// TwinCAT 3 PLC project PLC1
// ProgramVersion: 3.1.4023.0
// libraries:
//   Tc2_Standard, * (Beckhoff Automation GmbH)
//   Tc2_System, * (Beckhoff Automation GmbH)
//   Tc2_Utilities, * (Beckhoff Automation GmbH)
//   Tc3_IotBase, * (Beckhoff Automation GmbH)
//   Tc3_JsonXml, * (Beckhoff Automation GmbH)
//   Tc3_Module, * (Beckhoff Automation GmbH)
// project tree:
//   DUTs/ ST_INSUMOS.TcDUT (not stored)
//   / PlcTask.TcTTO (not stored)
//   POUs/ CheckBounds.TcPOU, CheckDivDInt.TcPOU (not stored), CheckDivLInt.TcPOU (not stored), CheckDivLReal.TcPOU, CheckDivReal.TcPOU (not stored), CheckLRangeSigned.TcPOU, CheckLRangeUnsigned.TcPOU, CheckPointer.TcPOU, CheckRangeSigned.TcPOU (not stored), CheckRangeUnsigned.TcPOU (not stored), MAIN.TcPOU
//   POUs/HTTP/ FB_ParseString.TcPOU (not stored), FB_TestHTTP_Get.TcPOU, FB_TestHTTP_HeaderAuth.TcPOU (not stored), FB_TestHTTP_Post.TcPOU (not stored), FB_TestHTTP_Put.TcPOU (not stored)

// ---- POUs/CheckBounds.TcPOU
// Implicitly generated code : DO NOT EDIT
FUNCTION CheckBounds : DINT
VAR_INPUT
	index, lower, upper: DINT;
END_VAR

// Implicitly generated code : Only an Implementation suggestion
{noflow}
IF  index < lower THEN
	CheckBounds := lower;
ELSIF  index > upper THEN
	CheckBounds := upper;
ELSE  
	CheckBounds := index;
END_IF
{flow}

END_FUNCTION

// ---- POUs/CheckDivLReal.TcPOU
// Implicitly generated code : DO NOT EDIT
FUNCTION CheckDivLReal : LREAL
VAR_INPUT
	divisor:LREAL;
END_VAR

// Implicitly generated code : Only an Implementation suggestion
{noflow}
IF divisor = 0 THEN
	CheckDivLReal:=1;
ELSE
	CheckDivLReal:=divisor;
END_IF;
{flow}

END_FUNCTION

// ---- POUs/CheckLRangeSigned.TcPOU
// Implicitly generated code : DO NOT EDIT
FUNCTION CheckLRangeSigned : LINT
VAR_INPUT
	value, lower, upper: LINT;
END_VAR

// Implicitly generated code : Only an Implementation suggestion
{noflow}
IF (value < lower) THEN
	CheckLRangeSigned := lower;
ELSIF(value > upper) THEN
	CheckLRangeSigned := upper;
ELSE
	CheckLRangeSigned := value;
END_IF

{flow}

END_FUNCTION

// ---- POUs/CheckLRangeUnsigned.TcPOU
// Implicitly generated code : DO NOT EDIT
FUNCTION CheckLRangeUnsigned : ULINT
VAR_INPUT
	value, lower, upper: ULINT;
END_VAR

// Implicitly generated code : Only an Implementation suggestion
{noflow}
IF (value < lower) THEN
	CheckLRangeUnsigned := lower;
ELSIF(value > upper) THEN
	CheckLRangeUnsigned := upper;
ELSE
	CheckLRangeUnsigned := value;
END_IF
{flow}

END_FUNCTION

// ---- POUs/CheckPointer.TcPOU
// Implicitly generated code : DO NOT EDIT
FUNCTION CheckPointer : POINTER TO BYTE
VAR_INPUT 
	ptToTest : POINTER TO BYTE; // Destination address of the pointer
	iSize : DINT;		        // Size of the type the pointer points to. (e.g: 20 for POINTER TO ARRAY [0..9] OF INT) 
	iGran : DINT;		        // Granularity of the pointer access. This is the size of the biggest non-structured data type in the type the pointer points to. (e.g: 2 for POINTER TO ARRAY [0..9] OF INT)
	bWrite: BOOL;		        // Indicates read or write Access. TRUE = write access.
END_VAR

// Implicitly generated code : Only an Implementation suggestion
{noflow}
IF ptToTest=0 THEN
    ADSLOGSTR(ADSLOG_MSGTYPE_ERROR OR ADSLOG_MSGTYPE_STRING,'CheckPointer failed due to invalid address.','');
ELSIF iSize<=0 THEN
    ADSLOGSTR(ADSLOG_MSGTYPE_ERROR OR ADSLOG_MSGTYPE_STRING,'CheckPointer failed due to invalid size.','');
ELSIF iGran<=0 THEN
    ADSLOGSTR(ADSLOG_MSGTYPE_ERROR OR ADSLOG_MSGTYPE_STRING,'CheckPointer failed due to invalid granularity.','');
// -> Please note that the following memory area check is time consuming:
//ELSIF F_CheckMemoryArea(pData:=ptToTest,nSize:=DINT_TO_UDINT(iSize)) = E_TcMemoryArea.Unknown THEN
//    ADSLOGSTR(ADSLOG_MSGTYPE_ERROR OR ADSLOG_MSGTYPE_STRING,'CheckPointer failed due to unknown memory area.','');
END_IF
CheckPointer := ptToTest;
{flow}

END_FUNCTION

// ---- POUs/MAIN.TcPOU
PROGRAM MAIN
VAR
	fbHttpClientPostman			: FB_IotHttpClient := (sHostName := '10.1.1.220',bKeepAlive:=TRUE);	
	fbHttpHeaderAuth			: FB_TestHTTP_HeaderAuth;
	
	bHeaderAuth 				: BOOL;
	bConvertBack				: BOOL;
	fbJsonDataType				: FB_JsonReadWriteDatatype;
	
	fbJson     : FB_JsonDomParser;
  		jsonProp   : SJsonValue;
  		jsonValue  : SJsonValue;
		
	bHasMember				: BOOL;
	operadorEncerrouLote	: DINT;
	data					: STRING(5000);
	insumos					: STRING(5000);
	arraySize				: UDINT;
	jsonIterator			: SJsonValue;
	jsonIteratorEnd			: SJsonValue;
	jsonIterator2			: SJsonValue;
	jsonIteratorEnd2		: SJsonValue;
	jsonIterator3			: SJsonValue;
	jsonIteratorEnd3		: SJsonValue;
	sName					: SJsonValue;
	jsonRoot				: SJsonValue;
	jsonRootInsumos			: SJsonValue;
	jsonRootInsumosDados	: SJsonValue;
	
	sTest:STRING(5000)		:= '{"continuationToken":"","data":[{"Insumos":[{"continuationToken":"","dados":[{"bloqueiaTerc":null,"centroCusto":"1011201002","classificacao":"1","classificacaoOrigem":"2","engenharia":"0201010080-0","insumo":"202010158","kanban":false,"natureza":"3","possuiAlternativos":false,"quantidadeTotal":"20000000","seqConsumo":4,"seqOperacao":1,"tipoInsumo":"1","transacaoBaixaEstoque":31},{"bloqueiaTerc":null,"centroCusto":"1011201002","classificacao":"1","classificacaoOrigem":"2","engenharia":"0201010080-0","insumo":"204010081","kanban":false,"natureza":"3","possuiAlternativos":false,"quantidadeTotal":"20000000","seqConsumo":2,"seqOperacao":1,"tipoInsumo":"1","transacaoBaixaEstoque":31},{"bloqueiaTerc":null,"centroCusto":"1011201002","classificacao":"1","classificacaoOrigem":"2","engenharia":"0201010080-0","insumo":"205050005","kanban":false,"natureza":"3","possuiAlternativos":false,"quantidadeTotal":"20000000","seqConsumo":3,"seqOperacao":1,"tipoInsumo":"1","transacaoBaixaEstoque":31}]}],"Lotes":[{"OperadorEncerrouLote":"163","codLote":"1-1","codOF":71605,"dadosLote":{"Operador":"","bloqueado":"","codLote":"1-1","codOF":71605,"dataHoraLiberacao":"","dataInicio":"2023-06-26","dataTermino":"2023-06-26","loteProducao":"0","motivo1":"","motivo2":"","quantidade":"100000"},"dataBaixa":"2023-06-26","dataBaixaRefugado":"","dataCancelamento":"","dataHoraEncerramento":"2023-06-26 15:43:33","dataHoraEncerramentoLote":"2023-06-26 15:43:33","dataTerminoTrefila":"","documento":"","observacao1":"","observacao2":"","observacao3":"","observacao4":"","operador":"","quantidade":"100000","quantidadeProd":"100000","quantidadeRefugo":"0","quantidadeUnd":"","quantidadeUndProd":"100000","quantidadeUndRefugo":"0","situacao":1,"tipo":""}],"Processos":[{"continuationToken":"","processos":[{"centroCustos":"1011201002","dadosCustomizados":[],"engenharia":"0201010080-0","faseProducao":4,"ferramentas":"","maquina":"10207010","numOperadores":"1","operacao":50,"sequencia":1,"tempoPadrao":"80","tempoPreparacao":"0","tipoOperacao":""}]}],"anoMes":202306,"codigoIntegracao":"","controle":"S-21911","dadosCustomizados":[],"dataInicio":"2023-06-26","dataTermino":"2023-06-26","finalidade":"","maquina":"","observacao1":"OF gerada pela simulacao nr. 21911.","observacao2":"","observacao3":"","observacao4":"","ordemFabricacao":"71605","planoProducao":"","produto":"0201010080-0","quantidade":"100000","semanaProducao":""}]}';

	i: INT;
	j: INT;
	
	arrInsumos 				: ARRAY[0..99] OF ST_INSUMOS;
	jsonProp2: SJsonValue;
	jsonProp3: SJsonValue;
	jsonProp4: SJsonValue;
	bBreak: BOOL;
END_VAR

// init client parameters at startup
IF NOT fbHttpClientPostman.bConfigured THEN 
	fbHttpClientPostman.stTLS.sCA 				 := 'C:\Users\PC042\Desktop\BECKHOFF\sample_cert.cer';
	fbHttpClientPostman.stTLS.bNoServerCertCheck := TRUE;
	fbHttpClientPostman.nHostPort				 := 443;
END_IF

IF fbHttpClientPostman.bConfigured THEN 
	fbHttpHeaderAuth(bSend:=bHeaderAuth, fbClient:=fbHttpClientPostman);
END_IF 

fbHttpClientPostman.Execute();

IF bConvertBack THEN
	jsonRoot:= fbJson.ParseDocument(sTest);	
	jsonProp := fbJson.FindMemberPath(jsonRoot, 'data');
	
	IF jsonProp <> 0 THEN
		jsonIterator := fbJson.ArrayBegin(jsonProp);
		jsonIteratorEnd := fbJson.ArrayEnd(jsonProp);
		WHILE jsonIterator <> jsonIteratorEnd DO
			fbJson.CopyJson(jsonIterator,data,SIZEOF(data));			
			jsonRootInsumos:= fbJson.ParseDocument(data);
			
			jsonProp2 := fbJson.FindMemberPath(jsonRootInsumos, 'Insumos');		
			fbJson.CopyJson(jsonProp2,data,SIZEOF(data));	
			
			IF jsonProp2 <> 0 THEN				
				jsonIterator2 := fbJson.ArrayBegin(jsonProp2);
				jsonIteratorEnd2 := fbJson.ArrayEnd(jsonProp2);
				WHILE jsonIterator2 <> jsonIteratorEnd2 DO	
						fbJson.CopyJson(jsonIterator2,data,SIZEOF(data));
						jsonRootInsumosDados:= fbJson.ParseDocument(data);
						
						jsonProp3 := fbJson.FindMemberPath(jsonRootInsumosDados, 'dados');
						fbJson.CopyJson(jsonProp3,data,SIZEOF(data));	
					
						IF jsonProp3 <> 0 THEN
							jsonIterator3 := fbJson.ArrayBegin(jsonProp3);
							jsonIteratorEnd3 := fbJson.ArrayEnd(jsonProp3);							
							WHILE (jsonIterator3 <> jsonIteratorEnd3) AND (NOT bBreak) DO
								fbJson.CopyJson(jsonIterator3,data,SIZEOF(data));
								
								jsonProp4 := fbJson.FindMember(jsonIterator3, 'bloqueiaTerc');										
								IF jsonProp4 <> 0 THEN
									arrInsumos[i].bBloqueiaTerc := fbJson.GetBool(jsonProp4);
								END_IF
								
								jsonProp4 := fbJson.FindMember(jsonIterator3, 'centroCusto');										
								IF jsonProp4 <> 0 THEN
									arrInsumos[i].sCentroCusto := fbJson.GetString(jsonProp4);
								END_IF								
								
								jsonProp4 := fbJson.FindMember(jsonIterator3, 'classificacao');										
								IF jsonProp4 <> 0 THEN
									arrInsumos[i].sClassificacao := fbJson.GetString(jsonProp4);
								END_IF
								
								jsonProp4 := fbJson.FindMember(jsonIterator3, 'classificacaoOrigem');										
								IF jsonProp4 <> 0 THEN
									arrInsumos[i].sClassificacaoOrigem := fbJson.GetString(jsonProp4);
								END_IF
								
								jsonProp4 := fbJson.FindMember(jsonIterator3, 'engenharia');										
								IF jsonProp4 <> 0 THEN
									arrInsumos[i].sEngenharia := fbJson.GetString(jsonProp4);
								END_IF
								
								jsonProp4 := fbJson.FindMember(jsonIterator3, 'insumo');										
								IF jsonProp4 <> 0 THEN
									arrInsumos[i].sInsumo := fbJson.GetString(jsonProp4);
								END_IF
								
								jsonProp4 := fbJson.FindMember(jsonIterator3, 'kanban');										
								IF jsonProp4 <> 0 THEN
									arrInsumos[i].bKanban := fbJson.GetBool(jsonProp4);
								END_IF
								
								jsonProp4 := fbJson.FindMember(jsonIterator3, 'natureza');										
								IF jsonProp4 <> 0 THEN
									arrInsumos[i].sNatureza := fbJson.GetString(jsonProp4);
								END_IF
								
								jsonProp4 := fbJson.FindMember(jsonIterator3, 'possuiAlternativos');										
								IF jsonProp4 <> 0 THEN
									arrInsumos[i].bPossuiAlternativos := fbJson.GetBool(jsonProp4);
								END_IF
								
								jsonProp4 := fbJson.FindMember(jsonIterator3, 'quantidadeTotal');										
								IF jsonProp4 <> 0 THEN
									arrInsumos[i].sQuantidadeTotal := fbJson.GetString(jsonProp4);
								END_IF
								
								jsonProp4 := fbJson.FindMember(jsonIterator3, 'seqConsumo');										
								IF jsonProp4 <> 0 THEN
									arrInsumos[i].iSeqConsumo := fbJson.GetInt(jsonProp4);
								END_IF
								
								jsonProp4 := fbJson.FindMember(jsonIterator3, 'seqOperacao');										
								IF jsonProp4 <> 0 THEN
									arrInsumos[i].iSeqOperacao := fbJson.GetInt(jsonProp4);
								END_IF
								
								jsonProp4 := fbJson.FindMember(jsonIterator3, 'tipoInsumo');										
								IF jsonProp4 <> 0 THEN
									arrInsumos[i].sTipoInsumo := fbJson.GetString(jsonProp4);
								END_IF
								
								jsonProp4 := fbJson.FindMember(jsonIterator3, 'transacaoBaixaEstoque');										
								IF jsonProp4 <> 0 THEN
									arrInsumos[i].iTransacaoBaixaEstoque := fbJson.GetInt(jsonProp4);
								END_IF								
								
								
								
								jsonIterator3 := fbJson.NextArray(jsonIterator3);
								i := i + 1;
							END_WHILE
						END_IF
						
						jsonIterator2 := fbJson.NextArray(jsonIterator2);
				END_WHILE	
			END_IF
			
			jsonIterator := fbJson.NextArray(jsonIterator);
		  END_WHILE
	  i := 0;
	END_IF	
	
	
	bConvertBack:=FALSE;
END_IF

END_PROGRAM

// ---- POUs/HTTP/FB_TestHTTP_Get.TcPOU
FUNCTION_BLOCK FB_TestHTTP_Get
VAR_INPUT
	bSend				: BOOL;
END_VAR
VAR_IN_OUT
	fbClient			: FB_IotHttpClient;
END_VAR
VAR_OUTPUT
	bBusy				: BOOL;
	bError				: BOOL;
END_VAR
VAR
	fbRequest			: FB_IotHttpRequest;
	fbJson				: FB_JsonDomParser;
	nState				: UDINT;
	RisingEdge			: R_TRIG;
	
	bGetContentResult	: BOOL;
	sContent			: STRING(511);
	
	bGetJsonResult		: BOOL;
	jsonDoc				: SJsonValue;
	jsonVal				: SJsonValue;
	sResultValue		: STRING;
	
	nReqCount			: UDINT;	
	nResCount			: UDINT;
	nValidResCount		: UDINT;
	nErrCount			: UDINT;
END_VAR

RisingEdge(CLK:= bSend );
CASE nState OF
0:	
	IF RisingEdge.Q THEN 
		IF fbRequest.SendRequest(sUri:='/api/ppcppadrao/v10/ordemFabricacao/71604', fbClient:=fbClient, eRequestType:=ETcIotHttpRequestType.HTTP_Get, 0, 0, 0) THEN				
			nState:= 1;
			nReqCount:= nReqCount+1;
			
			
			
			
			
			
			
			
			
			
			
			
			
			
			
			
			
			
			
			
			
			
			
			
			
			
			
			
			
			
			
			
			
			
			
			
			
			
			
			
			
			
			
			
			
			
			
			
			
			
			
			
			
			
			
			
			
			
			
			
			
			
			
			
			
			
			
			
			
			
			
			
			
			
			
			
			
			
			
			
			
			
			
			
			
			
			
			
			
			
			
			
			
			
			
			
			
			
			
			
			
			
			
			
			
			
			
			
			
			
			
			
			
			
			
			
			
			
			
			
			
			
			
			
			
			
			
			
			
			
			
			
			
			
			
			
			
			
			
			
			
			
			
			
			
			
			
			
			
			
			
			
			
			
			
			
			
			
			
			
			
			
			
			
			
			
			
			
			
			
			
			
			
			
			
			
			
			
			
			
			
			
			
			
			
			
			
			
			
			
			
			
			
			
			
			
			
			
			
			
			
			
			
			
			
			
			
			
			
			
			
			
			
			
			
			
			
			
			
			
			
			
			
			
			
			
			
			
			
			
			
			
			
			
			
			
			
			
			
			
			
			
			
			
			
			
			
			
			
			
			
			
			
			
			
			
			
			
			
			
			
			
			
			
			
			
			
			
			
			
			
			
			
			
			
			
			
			
			
			
			
			
			
			
			
			
			
			
			
			
			
			
			
			
			
			
			
			
			
			
			
			
			
			
			
			
			
			
			
			
			
			
			
			
			
			
			
			
			
			
			
			
			
			
			
			
			
			
			
			
			
			
			
			
			
			
			
			
			
			
			
			
			
			
			
			
			
			
			
			
			
			
			
			
			
			
			
			
			
			
			
			
			
			.__CATCH.__CATCH.__CATCH.__CATCH.__CATCH.__CATCH.__CATCH.__CATCH.__CATCH.__CATCH.__CATCH.__CATCH.__CATCH.__CATCH.__CATCH.__CATCH.__CATCH.__CATCH.__CATCH.__CATCH.__CATCH.__CATCH.__CATCH.__CATCH.__CATCH.__CATCH.__CATCH.
			bBusy:= TRUE;
			bError:= FALSE;
		END_IF
	END_IF
1:
	IF NOT fbRequest.bBusy THEN
		bError:= TRUE;
		IF NOT fbRequest.bError THEN				 
			bGetContentResult:= fbRequest.GetContent(pContent:= ADR(sContent), nContentSize:= SIZEOF(sContent), bSetNullTermination:= TRUE);
			IF fbRequest.nStatusCode >= 200 AND fbRequest.nStatusCode < 300 THEN
				bGetJsonResult:= FALSE;
				jsonDoc:= fbRequest.GetJsonDomContent(fbJson);
				IF jsonDoc <> 0 THEN
					bGetJsonResult:= TRUE;
					IF fbJson.HasMember(jsonDoc, 'args')  THEN
						jsonVal:= fbJson.FindMember(jsonDoc, 'args');
						IF fbJson.HasMember(jsonVal, 'foo2')  THEN
							jsonVal:= fbJson.FindMember(jsonVal, 'foo2');
							nValidResCount:= nValidResCount+1;
							bError:= FALSE;						
							IF fbJson.IsString(jsonVal) THEN							
								sResultValue:= fbJson.GetString(jsonVal);									
							END_IF
						END_IF		
					END_IF
				END_IF							
				nResCount:= nResCount+1;			
			END_IF
		END_IF
		nState:= 0;
		bBusy:= FALSE;
		IF bError THEN
			nErrCount:= nErrCount+1;
		END_IF
	END_IF  	
END_CASE

END_FUNCTION_BLOCK
